{attribute 'GeneratedUsingTerminal: EL9227-4433-0018'}
{attribute addProperty BoxType "EL9227-4433-0018"}
{attribute addProperty Id "StatusAT %I*Status_1D9409A420LoadAT %I*UINT2CurrentAT %I*UINT2Voltage_InAT %I*UINT2Voltage_OutAT %I*UINT2"}
{attribute addProperty CRC "2034905627"}
{attribute addProperty Size "28"}
TYPE OCP_Inputs_Channel_794A321B EXTENDS InputBase_8311D824 :
STRUCT
	{attribute addProperty Name "Status"}
	Status AT %I* : Status_1D9409A4;
	{attribute addProperty Name "Load"}
	Load AT %I* : UINT;
	{attribute addProperty Name "Current"}
	Current AT %I* : UINT;
	{attribute addProperty Name "Voltage_In"}
	Voltage_In AT %I* : UINT;
	{attribute addProperty Name "Voltage_Out"}
	Voltage_Out AT %I* : UINT;
END_STRUCT
END_TYPE

(* stored: Version 1.2.0.0, ProductVersion 3.1.4024.11
   DUT OCP_Inputs_Channel_794A321B: Id {98b131bf-77fb-477b-8909-2ccbadeea119} *)
